TYPE ST_MotionLinxAxisRecipe :
	STRUCT
		Velocity		: INT;
		Acceleration	: INT;
		Deceleration	: INT;	
		MaxSpeed		:UINT;
	END_STRUCT
END_TYPE

(* stored: Version 1.1.0.1, ProductVersion 3.1.4024.16
   DUT ST_MotionLinxAxisRecipe: Id {945967ad-13cc-4513-8758-7da7a9ffe14a} *)
